(* CODESYS project Visualization.vis.xml

Project tree, tasks and I/O mapping:
  visualisation Visualization
*)

// /Visualization
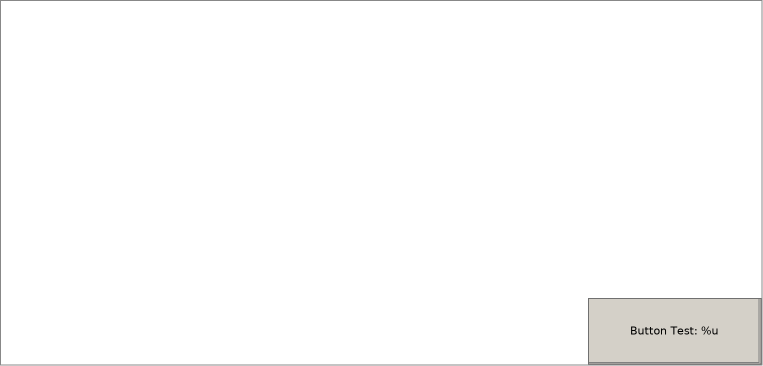
VISUALIZATION Visualization  // 763x366
    Button (588,298 173x66), "Button Test: %u", text variable: FB_TESTING.uiCurrSupplyVolt
END_VISUALIZATION
